RoboDK station: Sanding Station.rdk

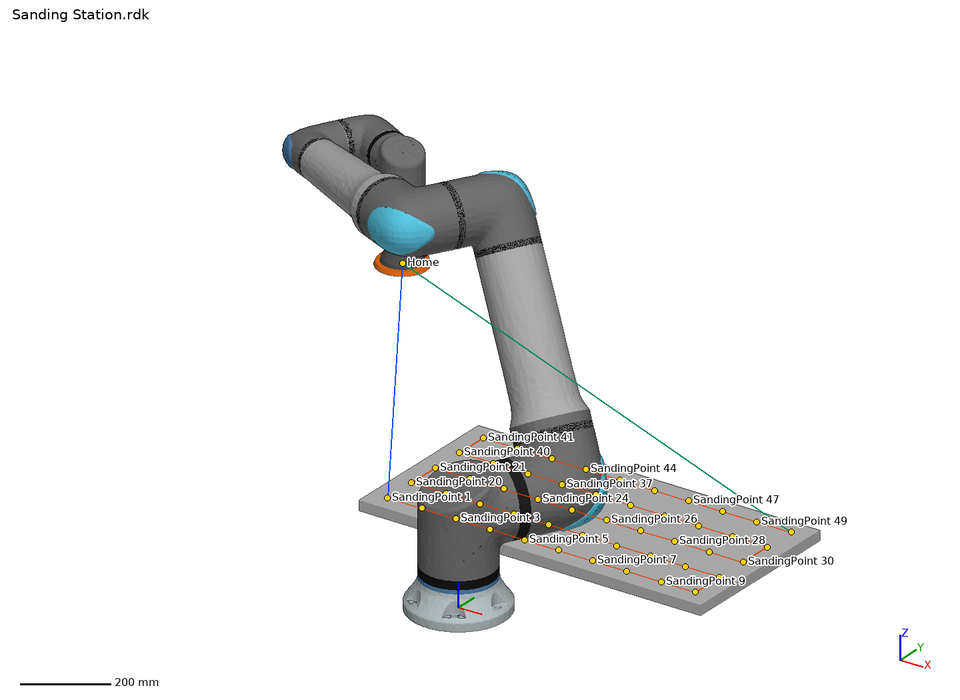
[picture v0: the station drawn from its stored meshes, robots at their saved joint values, targets as dots, program paths as lines]
Station Sanding Station (saved by RoboDK 5.7.1). Poses are relative to the parent item; angles as X-Y-Z fixed-axis rotations.
  - frame UR30 Base at (0, 0, 0) mm
    - robot UR30: 6 axes
        modified DH rows (alpha deg, a mm, theta deg, d mm): 0, 0, 0, 236.3; 90, 0, 0, 0; 0, 637, 0, 0; 0, 503.7, 0, 201; -90, 0, 0, 159.3; 90, 0, 180, 150
        joint limits [-360, -360, -360, -360, -360, -360] to [360, 360, 360, 360, 360, 360]; home [0, 90, -90, 0, 90, 0]; saved at [-208.486, 58.273, 297.388, -265.661, -90, -118.486]
      - tool RobotiQ Sanding Kit, TCP at (0, 0, 90) mm, size 139.7 x 127 x 103.3 mm
    - target Home (Cartesian target) at (-500, 500, 500) mm, rotated rx -180 ry 0 rz 0 deg; joints [-61.514, 94.06, 105.87, -109.93, -90, 28.486] of UR30
    - target SandingPoint 1 (Cartesian target) at (-411.48, 317.12, 25.4) mm, rotated rx 180 ry 0 rz 0 deg; joints [-194.858, 49.11, 246.959, -206.07, -90, -104.858] of UR30
    - target SandingPoint 2 (Cartesian target) at (-320.04, 317.12, 25.4) mm, rotated rx 180 ry 0 rz 0 deg; joints [-198.242, 52.116, 237.774, -199.89, -90, -108.242] of UR30
    - target SandingPoint 3 (Cartesian target) at (-228.6, 317.12, 25.4) mm, rotated rx 180 ry 0 rz 0 deg; joints [-203.272, 54.333, 229.822, -194.154, -90, -113.272] of UR30
    - target SandingPoint 4 (Cartesian target) at (-137.16, 317.12, 25.4) mm, rotated rx 180 ry 0 rz 0 deg; joints [-211.037, 55.695, 223.595, -189.29, -90, -121.037] of UR30
    - target SandingPoint 5 (Cartesian target) at (-45.72, 317.12, 25.4) mm, rotated rx -180 ry 0 rz 0 deg; joints [-222.942, 56.271, 220.01, -186.281, -90, -132.942] of UR30
    - target SandingPoint 6 (Cartesian target) at (45.72, 317.12, 25.4) mm, rotated rx 180 ry 0 rz 0 deg; joints [-239.35, 56.271, 220.01, -186.281, -90, -149.35] of UR30
    - target SandingPoint 7 (Cartesian target) at (137.16, 317.12, 25.4) mm, rotated rx -180 ry 0 rz 0 deg; joints [-257.816, 55.695, 223.595, -189.29, -90, -167.816] of UR30
    - target SandingPoint 8 (Cartesian target) at (228.6, 317.12, 25.4) mm, rotated rx 180 ry 0 rz 0 deg; joints [-274.845, 54.333, 229.822, -194.154, -90, -184.845] of UR30
    - target SandingPoint 9 (Cartesian target) at (320.04, 317.12, 25.4) mm, rotated rx -180 ry 0 rz 0 deg; joints [-288.767, 52.116, 237.774, -199.89, -90, -198.767] of UR30
    - target SandingPoint 10 (Cartesian target) at (411.48, 317.12, 25.4) mm, rotated rx 180 ry 0 rz 0 deg; joints [-299.617, 49.11, 246.959, -206.07, -90, -209.617] of UR30
    - target SandingPoint 11 (Cartesian target) at (411.48, 408.56, 25.4) mm, rotated rx 180 ry 0 rz 0 deg; joints [-294.922, 46.148, 255.181, -211.328, -90, -204.922] of UR30
    - target SandingPoint 12 (Cartesian target) at (320.04, 408.56, 25.4) mm, rotated rx -180 ry 0 rz 0 deg; joints [-285.287, 49.134, 246.89, -206.025, -90, -195.287] of UR30
    - target SandingPoint 13 (Cartesian target) at (228.6, 408.56, 25.4) mm, rotated rx 180 ry 0 rz 0 deg; joints [-273.803, 51.389, 240.112, -201.501, -90, -183.803] of UR30
    - target SandingPoint 14 (Cartesian target) at (137.16, 408.56, 25.4) mm, rotated rx -180 ry 0 rz 0 deg; joints [-260.757, 52.888, 235.175, -198.062, -90, -170.757] of UR30
    - target SandingPoint 15 (Cartesian target) at (45.72, 408.56, 25.4) mm, rotated rx -180 ry 0 rz 0 deg; joints [-247.116, 53.628, 232.529, -196.157, -90, -157.116] of UR30
    - target SandingPoint 16 (Cartesian target) at (-45.72, 408.56, 25.4) mm, rotated rx 180 ry 0 rz 0 deg; joints [-234.345, 53.628, 232.529, -196.157, -90, -144.345] of UR30
    - target SandingPoint 17 (Cartesian target) at (-137.16, 408.56, 25.4) mm, rotated rx -180 ry 0 rz 0 deg; joints [-223.642, 52.888, 235.175, -198.062, -90, -133.642] of UR30
    - target SandingPoint 18 (Cartesian target) at (-228.6, 408.56, 25.4) mm, rotated rx 180 ry 0 rz 0 deg; joints [-215.346, 51.389, 240.112, -201.501, -90, -125.346] of UR30
    - target SandingPoint 19 (Cartesian target) at (-320.04, 408.56, 25.4) mm, rotated rx -180 ry 0 rz 0 deg; joints [-209.141, 49.134, 246.89, -206.025, -90, -119.141] of UR30
    - target SandingPoint 20 (Cartesian target) at (-411.48, 408.56, 25.4) mm, rotated rx -180 ry 0 rz 0 deg; joints [-204.514, 46.148, 255.181, -211.328, -90, -114.514] of UR30
    - target SandingPoint 21 (Cartesian target) at (-411.48, 500, 25.4) mm, rotated rx 180 ry 0 rz 0 deg; joints [-212.463, 42.46, 264.794, -217.254, -90, -122.463] of UR30
    - target SandingPoint 22 (Cartesian target) at (-320.04, 500, 25.4) mm, rotated rx -180 ry 0 rz 0 deg; joints [-217.587, 45.429, 257.1, -212.528, -90, -127.587] of UR30
    - target SandingPoint 23 (Cartesian target) at (-228.6, 500, 25.4) mm, rotated rx 180 ry 0 rz 0 deg; joints [-223.986, 47.662, 251.052, -208.714, -90, -133.986] of UR30
    - target SandingPoint 24 (Cartesian target) at (-137.6, 500, 25.4) mm, rotated rx 180 ry 0 rz 0 deg; joints [-231.808, 49.153, 246.837, -205.99, -90, -141.808] of UR30
    - target SandingPoint 25 (Cartesian target) at (-45.72, 500, 25.4) mm, rotated rx 180 ry 0 rz 0 deg; joints [-241.177, 49.909, 244.627, -204.536, -90, -151.177] of UR30
    - target SandingPoint 26 (Cartesian target) at (45.72, 500, 25.4) mm, rotated rx -180 ry 0 rz 0 deg; joints [-251.626, 49.909, 244.627, -204.536, -90, -161.626] of UR30
    - target SandingPoint 27 (Cartesian target) at (137.16, 500, 25.4) mm, rotated rx 180 ry 0 rz 0 deg; joints [-262.53, 49.158, 246.821, -205.979, -90, -172.53] of UR30
    - target SandingPoint 28 (Cartesian target) at (228.6, 500, 25.4) mm, rotated rx 180 ry 0 rz 0 deg; joints [-273.125, 47.662, 251.052, -208.714, -90, -183.125] of UR30
    - target SandingPoint 29 (Cartesian target) at (320.04, 500, 25.4) mm, rotated rx -180 ry 0 rz 0 deg; joints [-282.832, 45.429, 257.1, -212.528, -90, -192.832] of UR30
    - target SandingPoint 30 (Cartesian target) at (411.48, 500, 25.4) mm, rotated rx 180 ry 0 rz 0 deg; joints [-291.37, 42.46, 264.794, -217.254, -90, -201.37] of UR30
    - target SandingPoint 31 (Cartesian target) at (411.48, 591.44, 25.4) mm, rotated rx -180 ry 0 rz 0 deg; joints [-288.628, 37.993, 275.894, -223.887, -90, -198.628] of UR30
    - target SandingPoint 32 (Cartesian target) at (320.04, 591.44, 25.4) mm, rotated rx -180 ry 0 rz 0 deg; joints [-281.027, 40.996, 268.484, -219.48, -90, -191.027] of UR30
    - target SandingPoint 33 (Cartesian target) at (228.6, 591.44, 25.4) mm, rotated rx -180 ry 0 rz 0 deg; joints [-272.651, 43.226, 262.838, -216.065, -90, -182.651] of UR30
    - target SandingPoint 34 (Cartesian target) at (137.16, 591.44, 25.4) mm, rotated rx -180 ry 0 rz 0 deg; joints [-263.723, 44.71, 258.993, -213.703, -90, -173.723] of UR30
    - target SandingPoint 35 (Cartesian target) at (45.72, 591.44, 25.4) mm, rotated rx -180 ry 0 rz 0 deg; joints [-254.614, 45.452, 257.037, -212.489, -90, -164.614] of UR30
    - target SandingPoint 36 (Cartesian target) at (-45.72, 591.44, 25.4) mm, rotated rx -180 ry 0 rz 0 deg; joints [-245.774, 45.452, 257.037, -212.489, -90, -155.774] of UR30
    - target SandingPoint 37 (Cartesian target) at (-137.16, 591.44, 25.4) mm, rotated rx -180 ry 0 rz 0 deg; joints [-237.61, 44.71, 258.993, -213.703, -90, -147.61] of UR30
    - target SandingPoint 38 (Cartesian target) at (-228.6, 591.44, 25.4) mm, rotated rx -180 ry 0 rz 0 deg; joints [-230.387, 43.226, 262.838, -216.065, -90, -140.387] of UR30
    - target SandingPoint 39 (Cartesian target) at (-320.04, 591.44, 25.4) mm, rotated rx -180 ry 0 rz 0 deg; joints [-224.19, 40.996, 268.484, -219.48, -90, -134.19] of UR30
    - target SandingPoint 40 (Cartesian target) at (-411.48, 591.44, 25.4) mm, rotated rx -180 ry 0 rz 0 deg; joints [-218.974, 37.993, 275.894, -223.887, -90, -128.974] of UR30
    - target SandingPoint 41 (Cartesian target) at (-411.48, 682.88, 25.4) mm, rotated rx -180 ry 0 rz 0 deg; joints [-224.326, 32.57, 288.893, -231.463, -90, -134.326] of UR30
    - target SandingPoint 42 (Cartesian target) at (-320.04, 682.88, 25.4) mm, rotated rx -180 ry 0 rz 0 deg; joints [-229.432, 35.723, 281.385, -227.108, -90, -139.432] of UR30
    - target SandingPoint 43 (Cartesian target) at (-228.6, 682.88, 25.4) mm, rotated rx 180 ry 0 rz 0 deg; joints [-235.284, 38.018, 275.835, -223.852, -90, -145.284] of UR30
    - target SandingPoint 44 (Cartesian target) at (-137.16, 682.88, 25.4) mm, rotated rx 180 ry 0 rz 0 deg; joints [-241.87, 39.525, 272.139, -221.664, -90, -151.87] of UR30
    - target SandingPoint 45 (Cartesian target) at (-45.72, 682.88, 25.4) mm, rotated rx 180 ry 0 rz 0 deg; joints [-249.091, 40.274, 270.285, -220.559, -90, -159.091] of UR30
    - target SandingPoint 46 (Cartesian target) at (45.72, 682.88, 25.4) mm, rotated rx -180 ry 0 rz 0 deg; joints [-256.752, 40.274, 270.285, -220.559, -90, -166.752] of UR30
    - target SandingPoint 47 (Cartesian target) at (137.16, 682.88, 25.4) mm, rotated rx 180 ry 0 rz 0 deg; joints [-264.584, 39.525, 272.139, -221.664, -90, -174.584] of UR30
    - target SandingPoint 48 (Cartesian target) at (228.6, 682.88, 25.4) mm, rotated rx 180 ry 0 rz 0 deg; joints [-272.301, 38.018, 275.835, -223.852, -90, -182.301] of UR30
    - target SandingPoint 49 (Cartesian target) at (320.04, 682.88, 25.4) mm, rotated rx -180 ry 0 rz 0 deg; joints [-279.653, 35.723, 281.385, -227.108, -90, -189.653] of UR30
    - target SandingPoint 50 (Cartesian target) at (411.48, 682.88, 25.4) mm, rotated rx -180 ry 0 rz 0 deg; joints [-286.469, 32.57, 288.893, -231.463, -90, -196.469] of UR30
  - object TableTop at (0, 500, 12.7) mm, size 914.4 x 457.2 x 25.4 mm, geometry from TableTop.stl
  - program ApproachMove (4 instructions, listed below)
  - program SandingPath (52 instructions, listed below)
  - program Retract (4 instructions, listed below)
  - program MainProgram (3 instructions, listed below)
  - Python program Prog5 (listed below)
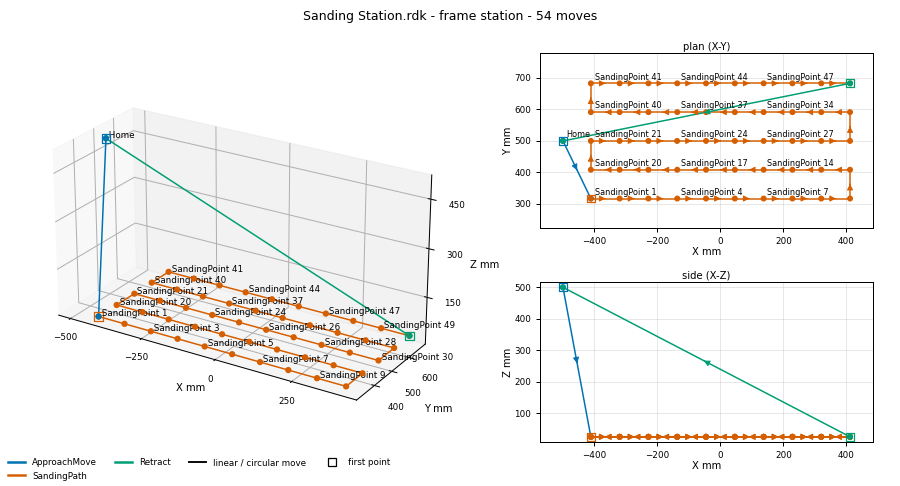
[picture p0: tool path of Sanding Station.rdk in frame station, 54 of 54 moves have a stored position in this frame; points joined in program order, loops and branches not executed]

--- program ApproachMove (robot UR30) ---
  Set Ref.: UR30 Base
  Set Tool: RobotiQ Sanding Kit
  MoveL (Home)
  MoveL (Target 2) -> target SandingPoint 1

--- program SandingPath (robot UR30) ---
  Set Ref.: UR30 Base
  Set Tool: RobotiQ Sanding Kit
  MoveJ (SandingPoint 1)
  MoveL (SandingPoint 2)
  MoveL (SandingPoint 3)
  MoveL (SandingPoint 4)
  MoveL (SandingPoint 5)
  MoveL (SandingPoint 6)
  MoveL (SandingPoint 7)
  MoveL (SandingPoint 8)
  MoveL (SandingPoint 9)
  MoveL (SandingPoint 10)
  MoveL (SandingPoint 11)
  MoveL (SandingPoint 12)
  MoveL (SandingPoint 13)
  MoveL (SandingPoint 14)
  MoveL (SandingPoint 15)
  MoveL (SandingPoint 16)
  MoveL (SandingPoint 17)
  MoveL (SandingPoint 18)
  MoveL (SandingPoint 19)
  MoveL (SandingPoint 20)
  MoveL (SandingPoint 21)
  MoveL (SandingPoint 22)
  MoveL (SandingPoint 23)
  MoveL (SandingPoint 24)
  MoveL (SandingPoint 25)
  MoveL (SandingPoint 26)
  MoveL (SandingPoint 27)
  MoveL (SandingPoint 28)
  MoveL (SandingPoint 29)
  MoveL (SandingPoint 30)
  MoveL (SandingPoint 31)
  MoveL (SandingPoint 32)
  MoveL (SandingPoint 33)
  MoveL (SandingPoint 34)
  MoveL (SandingPoint 35)
  MoveL (SandingPoint 36)
  MoveL (SandingPoint 37)
  MoveL (SandingPoint 38)
  MoveL (SandingPoint 39)
  MoveL (SandingPoint 40)
  MoveL (SandingPoint 41)
  MoveL (SandingPoint 42)
  MoveL (SandingPoint 43)
  MoveL (SandingPoint 44)
  MoveL (SandingPoint 45)
  MoveL (SandingPoint 46)
  MoveL (SandingPoint 47)
  MoveL (SandingPoint 48)
  MoveL (SandingPoint 49)
  MoveL (SandingPoint 50)

--- program Retract (robot UR30) ---
  Set Ref.: UR30 Base
  Set Tool: RobotiQ Sanding Kit
  MoveL (SandingPoint 50)
  MoveL (Home)

--- program MainProgram (robot UR30) ---
  Call ApproachMove
  Call SandingPath
  Call Retract

--- Python program Prog5 ---
# Type help("robodk.robolink") or help("robodk.robomath") for more information
# Press F5 to run the script
# Documentation: https://robodk.com/doc/en/RoboDK-API.html
# Reference:     https://robodk.com/doc/en/PythonAPI/robodk.html
# Note: It is not required to keep a copy of this file, your Python script is saved with your RDK project

# You can also use the new version of the API:
from robodk import robolink    # RoboDK API
from robodk import robomath    # Robot toolbox
RDK = robolink.Robolink()

# Forward and backwards compatible use of the RoboDK API:
# Remove these 2 lines to follow python programming guidelines
from robodk import *      # RoboDK API
from robolink import *    # Robot toolbox
# Link to RoboDK
# RDK = Robolink()

# Notify user:
print('To edit this program:\nright click on the Python program, then, select "Edit Python script"')

# Program example:
item = RDK.Item('base')
if item.Valid():
    print('Item selected: ' + item.Name())
    print('Item posistion: ' + repr(item.Pose()))

print('Items in the station:')
itemlist = RDK.ItemList()
print(itemlist)

# Provoking an exception will display the console output if you run this script from RoboDK
raise Exception('Program not edited.')
